(* IEC 61131-3 sources: CodesysTest/export/Unused/FB_SimBasicVacuum.pou, 2 files *)

(* ---- FB_SimBasicVacuum.pou.st ---- *)
(*#-#-#-#-#-#-#-#-#-#---Declaration---#-#-#-#-#-#-#-#-#-#-#-#-#*)

FUNCTION_BLOCK FB_SimBasicVacuum EXTENDS FB_BaseComponent IMPLEMENTS IVacuumBagOpen, IExecuteAutomatically
VAR_INPUT
	vacGrabDwell : REAL;
END_VAR
VAR_OUTPUT
END_VAR
VAR
	startVac : FB_SimulatedFeedback(name := CONCAT(_prefix,'Start Vac'));
END_VAR
(*#-#-#-#-#-#-#-#-#-#---Implementation---#-#-#-#-#-#-#-#-#-#-#-#-#*)

(* ---- ClearStatus.m.st ---- *)
(*#-#-#-#-#-#-#-#-#-#---Declaration---#-#-#-#-#-#-#-#-#-#-#-#-#*)

METHOD PRIVATE ClearStatus
VAR_INPUT
END_VAR
(*#-#-#-#-#-#-#-#-#-#---Implementation---#-#-#-#-#-#-#-#-#-#-#-#-#*)

startVac.in := FALSE;
THIS^.Execute();
